Fanuc KAREL source: kd00006.KL

PROGRAM KD00006
%STACKSIZE=65535
%PRIORITY=65535
VAR
I : INTEGER
J : INTEGER
B : BOOLEAN
R : REAL
S : STRING[80]
BEGIN
I=1
END KD00006
